// TwinCAT 3 PLC project PLC
// ProgramVersion: 3.1.4024.0
// libraries:
//   Tc2_DMX, * (Beckhoff Automation GmbH)
//   Tc2_Standard, * (Beckhoff Automation GmbH)
//   Tc2_System, * (Beckhoff Automation GmbH)
//   Tc3_Module, * (Beckhoff Automation GmbH)
// project tree:
//   / PlcTask.TcTTO
//   POUs/ MAIN_1.TcPOU, MAIN_1_1.TcPOU
// real-time tasks:
//   TASK PlcTask: cycle T#10ms, priority 20, ADS port 350
// I/O:
//   DEVICE Device 3 (EtherCAT), AmsNetId 192.168.0.150.4.1
//     Term 9 (EK1100) [EK1100 EtherCAT Coupler (2A E-Bus)]
//       Term 10 (EL6851) [EL6851 DMX Master]
//       Term 12 (EL9011) [EL9011 End Terminal]
//     Box 11 (EP3751-0160) [EP3751-0160 Acceleration Sensor]
// variable links:
//   PLC/PLC Instance <-> Device 3 (EtherCAT)/Box 11 (EP3751-0160)
//     PlcTask Inputs/MAIN_1.EP3751_0160_X <-> AI Acc X Inputs/Value
//     PlcTask Inputs/MAIN_1.EP3751_0160_Y <-> AI Acc Y Inputs/Value
//     PlcTask Inputs/MAIN_1.EP3751_0160_Z <-> AI Acc Z Inputs/Value
//   PLC/PLC Instance <-> Device 3 (EtherCAT)/Term 9 (EK1100)/Term 10 (EL6851)
//     PlcTask Inputs/MAIN_1.stEL6851InData/bCyclicTxDDisabled <-> DMX Status/Cyclic TxD disabled
//     PlcTask Inputs/MAIN_1.stEL6851InData/bDefaultDataSent <-> DMX Status/Default data sent
//     PlcTask Inputs/MAIN_1.stEL6851InData/bFrameSentToggle <-> DMX Status/Frame sent toggle
//     PlcTask Inputs/MAIN_1.stEL6851InData/bReceiveToggle <-> DMX Status/Receive toggle
//     PlcTask Inputs/MAIN_1.stEL6851InData/bTransmitAccepted <-> DMX Status/Transmit accepted
//     PlcTask Inputs/MAIN_1.stEL6851InData/bTxPDOToggle <-> DMX Status/TxPDO Toggle
//     PlcTask Inputs/MAIN_1.stEL6851InData/byStartCode <-> DMX Status/Start code
//     PlcTask Inputs/MAIN_1.stEL6851InData/wChannelLength <-> DMX Status/Channel length
//     PlcTask Outputs/MAIN_1.stEL6851OutData/arrData[{1..64}] <-> DMX Channel 1-64/Channel {1..64}  (64 links)
//     PlcTask Outputs/MAIN_1.stEL6851OutData/bDisableCyclicTxD <-> DMX Control/Disable cyclic TxD
//     PlcTask Outputs/MAIN_1.stEL6851OutData/bSendDefaultData <-> DMX Control/Send default data
//     PlcTask Outputs/MAIN_1.stEL6851OutData/bTransmitRequest <-> DMX Control/Transmit request
//     PlcTask Outputs/MAIN_1.stEL6851OutData/byStartCode <-> DMX Control/Start code
//     PlcTask Outputs/MAIN_1.stEL6851OutData/wChannelLength <-> DMX Control/Channel length

CONFIGURATION PLC
    RESOURCE PLC ON TwinCAT3
        TASK PlcTask(INTERVAL := T#10ms, PRIORITY := 20);
        PROGRAM MAIN_1 WITH PlcTask : MAIN_1;
    END_RESOURCE
END_CONFIGURATION

// ---- POUs/MAIN_1.TcPOU
PROGRAM MAIN_1
VAR CONSTANT
	DINT_Size:DINT :=2147483647;
	Byte_Size:DINT :=255;
END_VAR
VAR
	EP3751_0160_X AT%I*:DINT;
	EP3751_0160_Y AT%I*:DINT;
	EP3751_0160_Z AT%I*:DINT;
	
	
	
	stEL6851InData  AT%I*:  ST_EL6851InDataEx;
	stEL6851OutData AT%Q*: ST_EL6851OutData;
	stCommandBuffer : ST_DMXCommandBuffer;
	arrProcessData  : ARRAY [1..512] OF BYTE;
	
	fbDMX		: FB_EL6851CommunicationEx;
END_VAR


arrProcessData[1]:=TO_BYTE(LIMIT(0,(EP3751_0160_X*128/1100)+128,255));
arrProcessData[2]:=TO_BYTE(LIMIT(0,(EP3751_0160_Y*128/1100)+128,255));
arrProcessData[3]:=10;
arrProcessData[5]:=255;
arrProcessData[6]:=10;



fbDMX(
	wSourceManufacturerId:= 16#42_41, 
	dwSourceDeviceId:= 16#12_13_14_15, 
	bEnableSendingData:= TRUE, 
	bSetCycleMode:=TRUE , 
	bSendDefaultData:= , 
	uiDataLength:= 64 , 
	dwOptions:=  , 
	stEL6851InData:=	stEL6851InData , 
	stEL6851OutData:= 	stEL6851OutData, 
	stCommandBuffer:= 	stCommandBuffer, 
	arrProcessData:=	arrProcessData);

END_PROGRAM

// ---- POUs/MAIN_1_1.TcPOU
PROGRAM MAIN_1_1
VAR CONSTANT
	DINT_Size:DINT :=2147483647;
	Byte_Size:DINT :=255;
END_VAR
VAR
	EP3751_0160_X AT%I*:DINT;
	EP3751_0160_Y AT%I*:DINT;
	EP3751_0160_Z AT%I*:DINT;
	
	
	EP3751_0260_X AT%I*:DINT;
	EP3751_0260_Y AT%I*:DINT;
	EP3751_0260_Z AT%I*:DINT;	
	EP3751_0260_rX AT%I*:DINT;
	EP3751_0260_rY AT%I*:DINT;
	EP3751_0260_rZ AT%I*:DINT;
	
	
	stEL6851InData  AT%I*:  ST_EL6851InDataEx;
	stEL6851OutData AT%Q*: ST_EL6851OutData;
	stCommandBuffer : ST_DMXCommandBuffer;
	arrProcessData  : ARRAY [1..512] OF BYTE;
	
	fbDMX		: FB_EL6851CommunicationEx;
	fbSample	: TON;
	bEP3751_0160_active AT%I*:BOOL;
	aButtons	AT%I*: ARRAY [1..4] OF   BOOL;
	aLeds		AT%Q*: ARRAY [1..8] OF   BOOL;
	aTrig		: array[1..4] of r_trig;
	nIndex: INT;
	nState: INT:=2;
END_VAR

FOR nIndex:=1 TO 4 DO
	aTrig[nIndex](clk:=aButtons[nIndex]);
	IF aTrig[nIndex].Q  THEN
		IF  nState=nIndex THEN
			nState:=0; 
		ELSE
			nState:=nIndex;
		END_IF
	END_IF
END_FOR		

Memset(ADR(aLeds),0, SIZEOF(aLeds));

CASE nState OF 
	0: 	//No Control
		arrProcessData[1]:=0;
		arrProcessData[2]:=0;
		arrProcessData[3]:=0;
		arrProcessData[4]:=0;
		arrProcessData[5]:=0;
		arrProcessData[6]:=0;
		
	1: // Box without Gyro
		aLeds[1]:=TRUE;
		arrProcessData[1]:=TO_BYTE(LIMIT(0,(EP3751_0160_X*128/1100)+128,255));
		arrProcessData[2]:=TO_BYTE(LIMIT(0,(EP3751_0160_Y*128/1100)+128,255));
		arrProcessData[3]:=25;
		arrProcessData[5]:=255;
		arrProcessData[6]:=10;
		
		(*arrProcessData[1]:=TO_BYTE(LIMIT(0,(EP3751_0160_X*128/1100)+128,255));
		arrProcessData[2]:=TO_BYTE(LIMIT(0,(EP3751_0160_Y*128/1100)+128,255));
		arrProcessData[3]:=0;
		arrProcessData[5]:=0;
		arrProcessData[6]:=0;*)
		//arrProcessData[3]:=TO_BYTE((EP3751_0160_Z/DINT_Size)*256+128);
		//arrProcessData[1]:=LIMIT(0,TO_BYTE(arrProcessData[1]+(EP3751_0160_X/DINT_Size)),255);
		//arrProcessData[2]:=LIMIT(0,TO_BYTE(arrProcessData[2]+(EP3751_0160_Y/DINT_Size)),255);
		//arrProcessData[3]:=LIMIT(0,TO_BYTE(arrProcessData[3]+(EP3751_0160_Z/DINT_Size)),255);
		//arrProcessData[4]:=255;	
		
	2: // Box with Gyro
		aLeds[2]:=TRUE;
		arrProcessData[1]:=TO_BYTE(LIMIT(0,(EP3751_0160_X*128/1100)+128,255));
		arrProcessData[2]:=TO_BYTE(LIMIT(0,(EP3751_0160_Y*128/1100)+128,255));
		arrProcessData[3]:=10;
		arrProcessData[5]:=255;
		arrProcessData[6]:=10;
		
	3: // Box without Gyro and Color
		aLeds[3]:=TRUE;
		arrProcessData[1]:=TO_BYTE(LIMIT(0,(EP3751_0160_X*128/1100)+128,255));
		arrProcessData[2]:=TO_BYTE(LIMIT(0,(EP3751_0160_Y*128/1100)+128,255));
		arrProcessData[3]:=30;
		arrProcessData[5]:=255;
		arrProcessData[6]:=10;
		
	4: // Box with Gyro and Color
		aLeds[4]:=TRUE;
		arrProcessData[1]:=0;
		arrProcessData[2]:=0;
		arrProcessData[3]:=0;
		arrProcessData[4]:=0;
		arrProcessData[5]:=0;
		arrProcessData[6]:=0;
END_CASE


fbDMX(
	wSourceManufacturerId:= 16#42_41, 
	dwSourceDeviceId:= 16#12_13_14_15, 
	bEnableSendingData:= TRUE, 
	bSetCycleMode:=TRUE , 
	bSendDefaultData:= , 
	uiDataLength:= 64 , 
	dwOptions:=  , 
	stEL6851InData:=	stEL6851InData , 
	stEL6851OutData:= 	stEL6851OutData, 
	stCommandBuffer:= 	stCommandBuffer, 
	arrProcessData:=	arrProcessData);

END_PROGRAM
